FUNCTION_BLOCK ControlElevadorInicio
VAR_INPUT
		SFCreset:BOOL;
	    SeguridadOK : BOOL;
	    SensorArriba AT %I*: BOOL;
		SensorAbajo AT %I*:BOOL;
		Enabled AT %I*:BOOL;
		
		SensorPaletDentro AT %I*:BOOL;
		SensorPaletFuera AT %I*:BOOL;
		SensorPaletEnEspera AT %I*:BOOL;


		PulsadorBajar AT%I*: BOOL;
		PulsadorSubir AT%I*: BOOL;
		
		ResetError :BOOL;
		
		MotorElevacion_Status AT%I*:UINT;
		MotorExtraccion_Status AT%I*:UINT;

		PuedeExtraer :BOOL;
END_VAR
VAR_OUTPUT
		MotorElevacion_Freq  AT%Q*: UINT;
	    MotorElevacion_Command AT%Q*: INT;
		
		MotorExtraccion_Freq  AT%Q*: UINT;
	    MotorExtraccion_Command AT%Q*: INT;
		
		StopperOFF AT %Q*: BOOL;
		
		PresenciaCintaArriba AT%I* :BOOL;
		PresenciaCintaAbajo AT %I* : BOOL;	
		
		Ready: BOOL;
		EsperandoPalet :BOOL;
		
END_VAR
VAR
	VelocidadAlta :UINT := 4000;
	VelocidadBAJA :UINT := 1500;
	ModoVelocidadAlta :BOOL := FALSE;
	TiempoAltaVelocidad :TIME := T#3S;
	
	ERROR :BOOL;
	PosicionArriba: WORD := 141;

	HomeOk :BOOL;
END_VAR

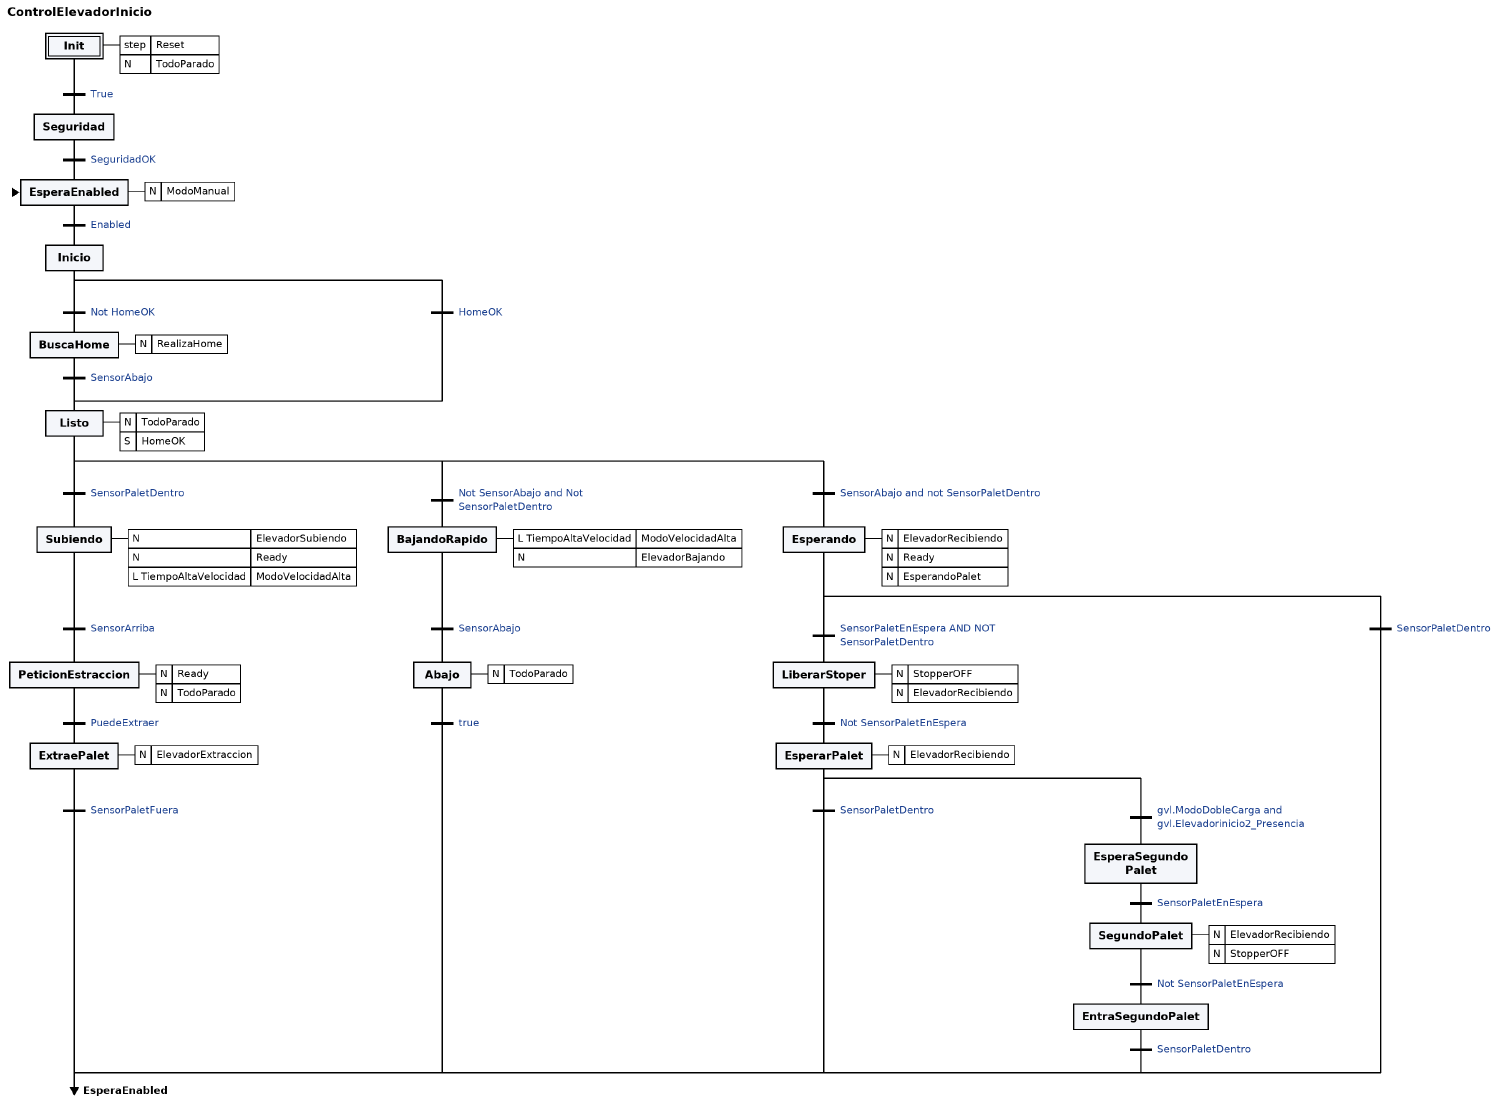
INITIAL_STEP Init:
    Reset(N);  // step action
    TodoParado(N);
END_STEP
TRANSITION FROM Init TO Seguridad
    := True;
END_TRANSITION
STEP Seguridad:
END_STEP
TRANSITION FROM Seguridad TO EsperaEnabled
    := SeguridadOK;
END_TRANSITION
STEP EsperaEnabled:
    ModoManual(N);
END_STEP
TRANSITION FROM EsperaEnabled TO Inicio
    := Enabled;
END_TRANSITION
STEP Inicio:
END_STEP
TRANSITION FROM Inicio TO BuscaHome
    := Not HomeOK;
END_TRANSITION
STEP BuscaHome:
    RealizaHome(N);
END_STEP
TRANSITION FROM BuscaHome TO Listo
    := SensorAbajo;
END_TRANSITION
TRANSITION FROM Inicio TO Listo
    := HomeOK;
END_TRANSITION
STEP Listo:
    TodoParado(N);
    HomeOK(S);
END_STEP
TRANSITION FROM Listo TO Subiendo
    := SensorPaletDentro;
END_TRANSITION
STEP Subiendo:
    ElevadorSubiendo(N);
    Ready(N);
    ModoVelocidadAlta(L, TiempoAltaVelocidad);
END_STEP
TRANSITION FROM Subiendo TO PeticionEstraccion
    := SensorArriba;
END_TRANSITION
STEP PeticionEstraccion:
    Ready(N);
    TodoParado(N);
END_STEP
TRANSITION FROM PeticionEstraccion TO ExtraePalet
    := PuedeExtraer;
END_TRANSITION
STEP ExtraePalet:
    ElevadorExtraccion(N);
END_STEP
TRANSITION FROM ExtraePalet TO EsperaEnabled
    := SensorPaletFuera;
END_TRANSITION
TRANSITION FROM Listo TO BajandoRapido
    := Not SensorAbajo and Not SensorPaletDentro;
END_TRANSITION
STEP BajandoRapido:
    ModoVelocidadAlta(L, TiempoAltaVelocidad);
    ElevadorBajando(N);
END_STEP
TRANSITION FROM BajandoRapido TO Abajo
    := SensorAbajo;
END_TRANSITION
STEP Abajo:
    TodoParado(N);
END_STEP
TRANSITION FROM Abajo TO EsperaEnabled
    := true;
END_TRANSITION
TRANSITION FROM Listo TO Esperando
    := SensorAbajo and not SensorPaletDentro;
END_TRANSITION
STEP Esperando:  // min time T#1s
    ElevadorRecibiendo(N);
    Ready(N);
    EsperandoPalet(N);
END_STEP
TRANSITION FROM Esperando TO LiberarStoper
    := SensorPaletEnEspera AND NOT SensorPaletDentro;
END_TRANSITION
STEP LiberarStoper:
    StopperOFF(N);
    ElevadorRecibiendo(N);
END_STEP
TRANSITION FROM LiberarStoper TO EsperarPalet
    := Not SensorPaletEnEspera;
END_TRANSITION
STEP EsperarPalet:
    ElevadorRecibiendo(N);
END_STEP
TRANSITION FROM EsperarPalet TO EsperaEnabled
    := SensorPaletDentro;
END_TRANSITION
TRANSITION FROM EsperarPalet TO EsperaSegundoPalet
    := gvl.ModoDobleCarga and gvl.Elevadorinicio2_Presencia;
END_TRANSITION
STEP EsperaSegundoPalet:
END_STEP
TRANSITION FROM EsperaSegundoPalet TO SegundoPalet
    := SensorPaletEnEspera;
END_TRANSITION
STEP SegundoPalet:
    ElevadorRecibiendo(N);
    StopperOFF(N);
END_STEP
TRANSITION FROM SegundoPalet TO EntraSegundoPalet
    := Not SensorPaletEnEspera;
END_TRANSITION
STEP EntraSegundoPalet:
END_STEP
TRANSITION FROM EntraSegundoPalet TO EsperaEnabled
    := SensorPaletDentro;
END_TRANSITION
TRANSITION FROM Esperando TO EsperaEnabled
    := SensorPaletDentro;
END_TRANSITION

ACTION ElevadorBajando:
MotorElevador(2);
MotorExtraccion(0);
END_ACTION

ACTION ElevadorExtraccion:

IF PuedeExtraer THEN
	MotorExtraccion(1);
ELSE 
	MotorExtraccion(0);
END_IF
END_ACTION

ACTION ElevadorRecibiendo:
MotorElevador(0);

IF Enabled THEN
	MotorExtraccion(2);
ELSE 
	MotorExtraccion(0);
END_IF
END_ACTION

ACTION ElevadorSubiendo:
MotorElevador(1);
MotorExtraccion(0);
END_ACTION

ACTION ModoManual:

IF PulsadorSubir THEN
		MotorElevador(1);
		HomeOK :=FALSE;
ELSIF PulsadorBajar THEN
		MotorElevador(2);
		HomeOK :=FALSE;
ELSE
		MotorElevador(0);	
END_IF
END_ACTION

METHOD PRIVATE MotorElevador : BOOL
VAR_INPUT
	Direccion : INT; //0 parado 1 subir 2 bajar
END_VAR
IF ModoVelocidadAlta THEN
	MotorElevacion_Freq := 5000;
ELSE
	MotorElevacion_Freq := 1000;
END_IF


MotorElevacion_Command := 0;
MotorElevacion_Command.7 := 1 ; //Control Word Active

IF Direccion = 0 THEN
	MotorElevacion_Command.3 := 1 ; // Stop according to parameter setting	
ELSIF PresenciaCintaArriba OR PresenciaCintaAbajo THEN
	//ERROR: intenta mover elevador con obstatuclos
	//DEBE MOStrar error
	MotorElevacion_Command.3 := 1 ; // Stop according to parameter setting	
ELSIF Direccion  = 1 THEN
	MotorElevacion_Command.2 := 0 ; //1 reversed 0 fordward
	MotorElevacion_Command.0 := 1 ; // Run Command active
		HomeOK :=FALSE;
ELSIF Direccion= 2 THEN
	MotorElevacion_Command.2 := 1 ; //1 reversed 0 fordward
	MotorElevacion_Command.0 := 1 ; // Run Command active
		HomeOK :=FALSE;
ELSE
	MotorElevacion_Command.3 := 1 ; // Stop according to parameter setting	
END_IF
END_METHOD

METHOD PRIVATE MotorExtraccion : BOOL
VAR_INPUT
	Direccion : INT; //0 parado 1 salida 2 entrada
END_VAR

MotorExtraccion_Freq := gvl.VelocidadCinta * 100;
MotorExtraccion_Command := 0;
MotorExtraccion_Command.7 := 1 ; //Control Word Active

IF Direccion  = 1 THEN
	MotorExtraccion_Command.2 := 0 ; //1 reversed 0 fordward
	MotorExtraccion_Command.0 := 1 ; // Run Command active
ELSIF Direccion= 2 THEN
	MotorExtraccion_Command.2 := 1 ; //1 reversed 0 fordward
	MotorExtraccion_Command.0 := 1 ; // Run Command active
ELSE
	MotorExtraccion_Command.3 := 1 ; // Stop according to parameter setting	
END_IF
END_METHOD

ACTION RealizaHome:
MotorElevador(2);
MotorExtraccion(0);
END_ACTION

ACTION Reset:
HomeOK := FALSE;
SFCreset:=FALSE;
END_ACTION

ACTION TodoParado:
MotorElevador(0);
MotorExtraccion(0);
END_ACTION

END_FUNCTION_BLOCK

(* stored: Version 1.1.0.1, ProductVersion 3.1.4024.3
   POU ControlElevadorInicio: Id {8be08686-48b7-4d87-aa9f-a90998bdba65}, SpecialFunc None
   Action ElevadorBajando: Id {ea8b950e-da8e-44a7-b583-0dab463ab183}
   Action ElevadorExtraccion: Id {f33005f7-1dd4-48c1-babd-523e8385f7f2}
   Action ElevadorRecibiendo: Id {7d3d520a-1072-4abc-a22c-6bed56447fb4}
   Action ElevadorSubiendo: Id {74046bd6-1b9d-4092-ad30-52f09f53d70e}
   Action ModoManual: Id {8f0e1d6e-52a3-42a9-869d-12658eedb19d}
   Method MotorElevador: Id {8297ddf0-046c-4dbb-b8a1-2c967404f2f4}
   Method MotorExtraccion: Id {b5da50e1-ac5e-4412-bcfc-f8675ab917ed}
   Action RealizaHome: Id {6ec733c1-473f-43fd-bfa2-e2ae0a44817a}
   Action Reset: Id {665761c2-a2f6-4db9-93b3-7b36fbcc3669}
   Action TodoParado: Id {a8e1dc7f-3903-43b3-b2ab-c6abce64c0b6} *)
